SUBAPPLICATION Uebung_160b2 (* Motor Links/Rechtslauf Automatisierung IX *)
  (* Standard: 61499-2; Description: Copyright (c) 2023 Meisterschulen am Ostbahnhof This program and the accompanying materials are made available under the terms of the Eclipse Public License 2.0 which is available at https://www.eclipse.org/legal/epl-2.0/ SPDX-License-Identifier: EPL-2.0 *)
  (* Version 1.0, 2023-10-23, Franz Höpfinger, Meisterschulen am Ostbahnhof, initial API and implementation and/or initial documentation *)
  PACKAGE Uebungen;
  IMPORT logiBUS::io::DI::logiBUS_DI::Input_I1;
  IMPORT logiBUS::io::DI::logiBUS_DI::Input_I2;
  IMPORT logiBUS::io::DI::logiBUS_DI::Input_I3;
  IMPORT logiBUS::io::DQ::logiBUS_DO::Output_Q5;
  IMPORT logiBUS::io::DQ::logiBUS_DO::Output_Q56;
  IMPORT logiBUS::io::DQ::logiBUS_DO::Output_Q6;
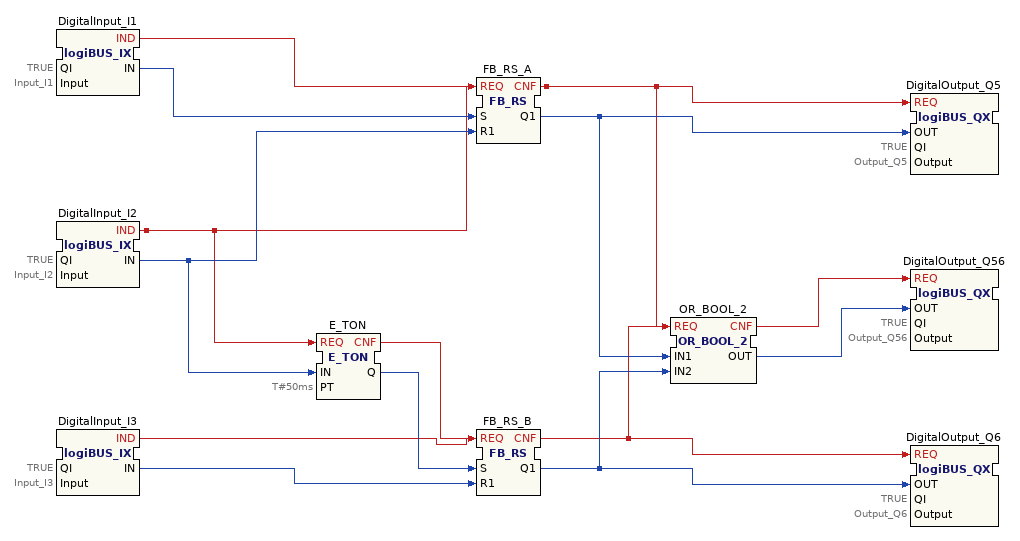
  FBS
    DigitalOutput_Q6 : logiBUS::io::DQ::logiBUS_QX(QI := TRUE, Output := Output_Q6);
    FB_RS_B : iec61131::bistableElements::FB_RS;
    OR_BOOL_2 : iec61131::booleanOperators::OR_BOOL_2;
    FB_RS_A : iec61131::bistableElements::FB_RS;
    DigitalOutput_Q5 : logiBUS::io::DQ::logiBUS_QX(QI := TRUE, Output := Output_Q5);
    DigitalOutput_Q56 : logiBUS::io::DQ::logiBUS_QX(QI := TRUE, Output := Output_Q56);
    DigitalInput_I2 : logiBUS::io::DI::logiBUS_IX(QI := TRUE, Input := Input_I2);
    DigitalInput_I3 : logiBUS::io::DI::logiBUS_IX(QI := TRUE, Input := Input_I3);
    DigitalInput_I1 : logiBUS::io::DI::logiBUS_IX(QI := TRUE, Input := Input_I1);
    E_TON : iec61499::events::timers::E_TON(PT := T#50ms);
  END_FBS
  EVENT_CONNECTIONS
    FB_RS_B.CNF TO DigitalOutput_Q6.REQ;
    FB_RS_A.CNF TO DigitalOutput_Q5.REQ;
    OR_BOOL_2.CNF TO DigitalOutput_Q56.REQ;
    FB_RS_B.CNF TO OR_BOOL_2.REQ;
    FB_RS_A.CNF TO OR_BOOL_2.REQ;
    DigitalInput_I2.IND TO E_TON.REQ;
    E_TON.CNF TO FB_RS_B.REQ;
    DigitalInput_I3.IND TO FB_RS_B.REQ;
    DigitalInput_I1.IND TO FB_RS_A.REQ;
    DigitalInput_I2.IND TO FB_RS_A.REQ;
  END_CONNECTIONS
  DATA_CONNECTIONS
    FB_RS_B.Q1 TO DigitalOutput_Q6.OUT;
    FB_RS_A.Q1 TO DigitalOutput_Q5.OUT;
    OR_BOOL_2.OUT TO DigitalOutput_Q56.OUT;
    FB_RS_A.Q1 TO OR_BOOL_2.IN1;
    FB_RS_B.Q1 TO OR_BOOL_2.IN2;
    E_TON.Q TO FB_RS_B.S;
    DigitalInput_I2.IN TO E_TON.IN;
    DigitalInput_I3.IN TO FB_RS_B.R1;
    DigitalInput_I1.IN TO FB_RS_A.S;
    DigitalInput_I2.IN TO FB_RS_A.R1;
  END_CONNECTIONS
END_SUBAPPLICATION
